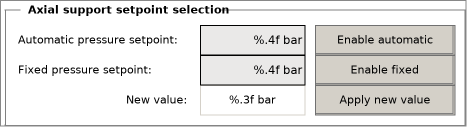
VISUALIZATION VISU_M1AxialSupportSetpoint  // 467x127
VAR_IN_OUT
	ref : M1AxialSupport;
    widget : M1AxialSupportWidget;
END_VAR
    Polyline (20,10) (5,10) (5,125) (465,125) (465,10) (220,10)
    Label (15,25 185x30), "Automatic pressure setpoint:"
    Label (15,55 185x30), "Fixed pressure setpoint:"
    Rectangle (200,25 105x30), "%.4f bar", text variable: ref.autoPressureSetpoint.bar.value
    Textfield (200,85 105x30), "%.3f bar", text variable: ref.processes.changePressureSetpoint.set.setpoint, input disabled if: ref.processes.changePressureSetpoint.statuses.enabledStatus.disabled
        OnMouseClick: write the text variable via Default
    Button (315,25 140x30), "Enable automatic", input disabled if: widget.changeToAutoButtonDeactivated
        OnMouseClick: execute { ref.processes.changePressureSetpointState.set.state := OperatingStates.AUTO; ref.processes.changePressureSetpointState.do_request := TRUE; }
    Button (315,55 140x30), "Enable fixed", input disabled if: widget.changeToManualButtonDeactivated
        OnMouseClick: execute { ref.processes.changePressureSetpointState.set.state := OperatingStates.MANUAL; ref.processes.changePressureSetpointState.do_request := TRUE; }
    Label (25,0 200x20), "Axial support setpoint selection"
    Button (315,85 140x30), "Apply new value", input disabled if: ref.processes.changePressureSetpoint.statuses.enabledStatus.disabled
        OnMouseClick: execute { ref.processes.changePressureSetpoint.do_request := TRUE; }
    Label (75,85 115x30), "New value:"
    Rectangle (200,55 105x30), "%.4f bar", text variable: ref.manualPressureSetpoint.bar.value
END_VISUALIZATION

(* stored: Version 1.1.0.1, ProductVersion 3.1.4018.2
   Visu VISU_M1AxialSupportSetpoint: Id {87f9cad9-62ea-4200-a7b5-34e7100288ae} *)
